FUNCTION_BLOCK Button_LS (* Composite Function Block Type *)
  (* Standard: 61499-2 *)
  (* Version 0.0, 07/03/2023, Pranay Jhunjhunwala, nxtControl GmBH, template *)
  PACKAGE Main;
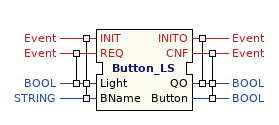
  EVENT_INPUT
    INIT WITH BName, Light; (* Initialization Request *)
    REQ WITH Light; (* Normal Execution Request *)
  END_EVENT
  EVENT_OUTPUT
    INITO WITH QO; (* Initialization Confirm *)
    CNF WITH QO, Button; (* Execution Confirmation *)
  END_EVENT
  VAR_INPUT
    Light : BOOL;
    BName : STRING;
  END_VAR
  VAR_OUTPUT
    QO : BOOL; (* Output event qualifier *)
    Button : BOOL;
  END_VAR
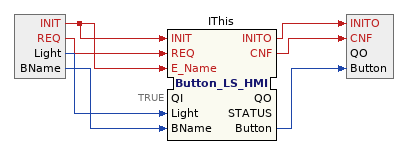
  FBS
    IThis : Button_LS_HMI(QI := TRUE);
  END_FBS
  EVENT_CONNECTIONS
    INIT TO IThis.INIT;
    REQ TO IThis.REQ;
    INIT TO IThis.E_Name;
    IThis.INITO TO INITO;
    IThis.CNF TO CNF;
  END_CONNECTIONS
  DATA_CONNECTIONS
    Light TO IThis.Light;
    BName TO IThis.BName;
    IThis.Button TO Button;
  END_CONNECTIONS
END_FUNCTION_BLOCK
